// TIA Portal V18 export
FUNCTION_BLOCK "02_Safety_Door"   // FB5, F_LAD
{ S7_Optimized_Access := 'TRUE' }
   VAR_INPUT
      Bypass_For_Commissioning : Bool;
      DIAG : Bool := TRUE;
      CH1 : Bool := TRUE;
      CH2 : Bool := TRUE;
      "Sorter_Running_from MSC" : Bool;
      Sorter_Stop_from_Encoder : Bool;
      Open_Request : Bool;
      Alarm_Filter : Bool;
      Sorter_Door : Bool := TRUE;   // If =1 sorter door management, if =0 management via ESTOP
      ACK_NEC : Bool := TRUE;   // If =1 door need to be reset, if = 0 door will autoreset
      ACK : Bool;
      ON_Lamp : Bool := TRUE;   // If = 1 reset lamp management, if = 0 reset lamp not present
   END_VAR
   VAR_OUTPUT
      Solenoid : Bool;
      EM_Cut : Bool;
      EM_Cut_Delay : Bool;
      Diag_Open : Bool;
      Diag_Alarm : Bool;
      Reset_Lamp : Bool;
   END_VAR
   VAR
      "E-STOP" : ESTOP1;
      TON_Alarm : TON;
      TOF_DoorLamp : TOF;
   END_VAR
   VAR_TEMP
      Alarm_Temp : Bool;
      t_ALARM : Bool;
      t_Lamp : Bool;
   END_VAR
   VAR CONSTANT
      Blink_Cycle_Time : Time := T#1S_260MS;
      ON_Time : Time := T#630MS;
   END_VAR
BEGIN

REGION Network 1: Emergency cut
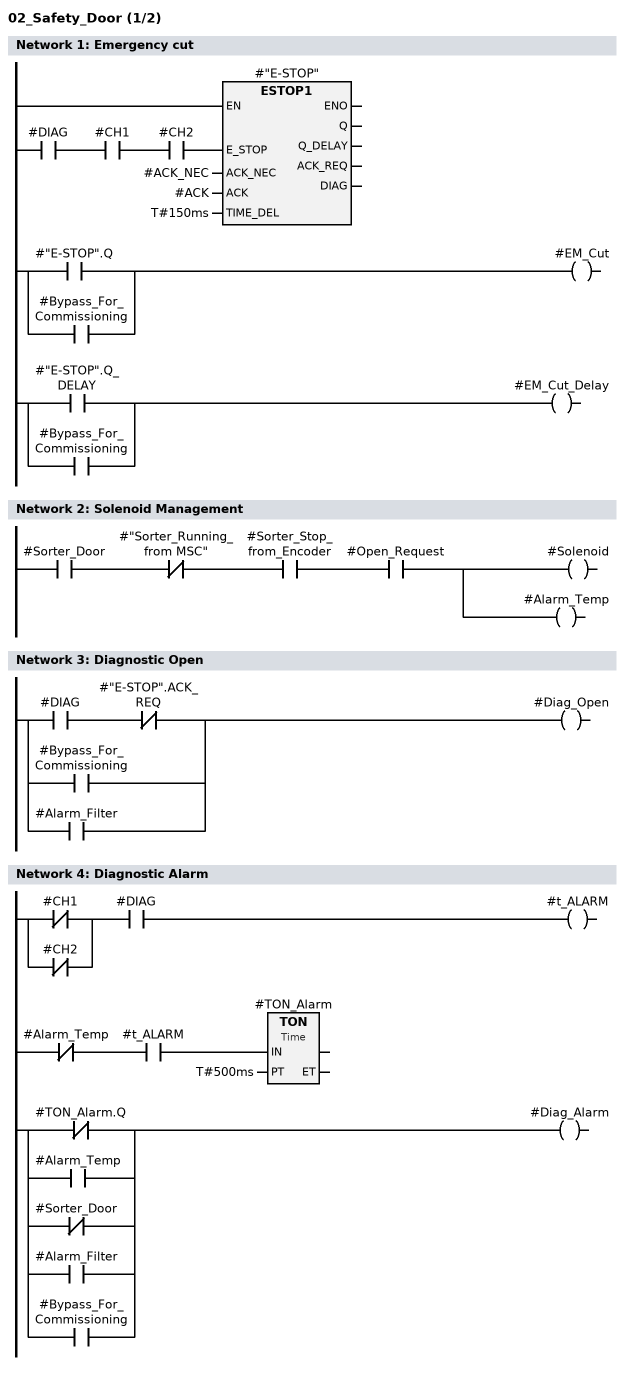
   RUNG wire#powerrail
      #"E-STOP".ESTOP1(E_STOP := wire#w1, ACK_NEC := #ACK_NEC, ACK := #ACK, TIME_DEL := T#150ms, Q =>, Q_DELAY =>, ACK_REQ =>, DIAG =>)
   END_RUNG
   RUNG wire#powerrail
      Contact( #DIAG )
      Contact( #CH1 )
      Contact( #CH2 )
   END_RUNG wire#w1
   RUNG wire#powerrail
      Contact( #"E-STOP".Q )
      wire#w2
      Coil( #EM_Cut )
   END_RUNG
   RUNG wire#powerrail
      Contact( #Bypass_For_Commissioning )
   END_RUNG wire#w2
   RUNG wire#powerrail
      Contact( #"E-STOP".Q_DELAY )
      wire#w3
      Coil( #EM_Cut_Delay )
   END_RUNG
   RUNG wire#powerrail
      Contact( #Bypass_For_Commissioning )
   END_RUNG wire#w3
   // the same network as SCL:
   #"E-STOP"(E_STOP := #DIAG AND #CH1 AND #CH2, ACK_NEC := #ACK_NEC, ACK := #ACK, TIME_DEL := T#150ms);   // ESTOP1
   #EM_Cut := #"E-STOP".Q OR #Bypass_For_Commissioning;
   #EM_Cut_Delay := #"E-STOP".Q_DELAY OR #Bypass_For_Commissioning;
END_REGION

REGION Network 2: Solenoid Management
   RUNG wire#powerrail
      Contact( #Sorter_Door )
      I_Contact( #"Sorter_Running_from MSC" )
      Contact( #Sorter_Stop_from_Encoder )
      Contact( #Open_Request )
      wire#w1
      Coil( #Solenoid )
   END_RUNG
   RUNG wire#w1
      Coil( #Alarm_Temp )
   END_RUNG
   // the same network as SCL:
   #Solenoid := #Sorter_Door AND NOT #"Sorter_Running_from MSC" AND #Sorter_Stop_from_Encoder AND #Open_Request;
   #Alarm_Temp := #Solenoid;
END_REGION

REGION Network 3: Diagnostic Open
   RUNG wire#powerrail
      Contact( #DIAG )
      I_Contact( #"E-STOP".ACK_REQ )
      wire#w1
      Coil( #Diag_Open )
   END_RUNG
   RUNG wire#powerrail
      Contact( #Bypass_For_Commissioning )
   END_RUNG wire#w1
   RUNG wire#powerrail
      Contact( #Alarm_Filter )
   END_RUNG wire#w1
   // the same network as SCL:
   #Diag_Open := (#DIAG AND NOT #"E-STOP".ACK_REQ) OR #Bypass_For_Commissioning OR #Alarm_Filter;
END_REGION

REGION Network 4: Diagnostic Alarm
   RUNG wire#powerrail
      I_Contact( #CH1 )
      wire#w1
      Contact( #DIAG )
      Coil( #t_ALARM )
   END_RUNG
   RUNG wire#powerrail
      I_Contact( #CH2 )
   END_RUNG wire#w1
   RUNG wire#powerrail
      I_Contact( #Alarm_Temp )
      Contact( #t_ALARM )
      { S7_Templates := "[time_type := Time, codedbool_type := DInt]" } #TON_Alarm.TON(pt := T#500ms, et =>)
   END_RUNG
   RUNG wire#powerrail
      I_Contact( #TON_Alarm.Q )
      wire#w2
      Coil( #Diag_Alarm )
   END_RUNG
   RUNG wire#powerrail
      Contact( #Alarm_Temp )
   END_RUNG wire#w2
   RUNG wire#powerrail
      I_Contact( #Sorter_Door )
   END_RUNG wire#w2
   RUNG wire#powerrail
      Contact( #Alarm_Filter )
   END_RUNG wire#w2
   RUNG wire#powerrail
      Contact( #Bypass_For_Commissioning )
   END_RUNG wire#w2
   // the same network as SCL:
   #t_ALARM := (NOT #CH1 OR NOT #CH2) AND #DIAG;
   #TON_Alarm.TON(IN := NOT #Alarm_Temp AND #t_ALARM, PT := T#500ms);
   #Diag_Alarm := NOT #TON_Alarm.Q OR #Alarm_Temp OR NOT #Sorter_Door OR #Alarm_Filter OR #Bypass_For_Commissioning;
END_REGION

REGION Network 5: Rest Lamp
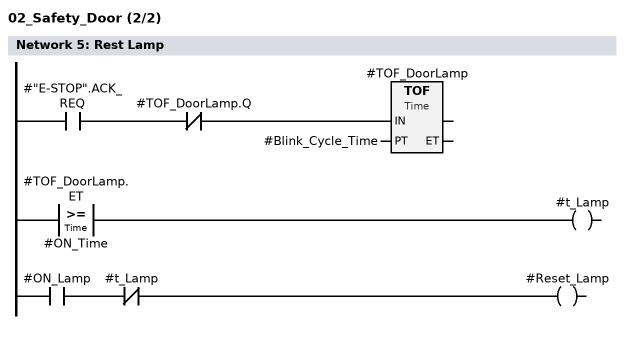
   RUNG wire#powerrail
      Contact( #"E-STOP".ACK_REQ )
      I_Contact( #TOF_DoorLamp.Q )
      { S7_Templates := "[time_type := Time, codedbool_type := DInt]" } #TOF_DoorLamp.TOF(pt := #Blink_Cycle_Time, et =>)
   END_RUNG
   RUNG wire#powerrail
      { S7_Templates := "SrcType := Time" } GE_Contact(in1 := #TOF_DoorLamp.ET, in2 := #ON_Time)
      Coil( #t_Lamp )
   END_RUNG
   RUNG wire#powerrail
      Contact( #ON_Lamp )
      I_Contact( #t_Lamp )
      Coil( #Reset_Lamp )
   END_RUNG
   // the same network as SCL:
   #TOF_DoorLamp.TOF(IN := #"E-STOP".ACK_REQ AND NOT #TOF_DoorLamp.Q, PT := #Blink_Cycle_Time);
   #t_Lamp := #TOF_DoorLamp.ET >= #ON_Time;
   #Reset_Lamp := #ON_Lamp AND NOT #t_Lamp;
END_REGION
END_FUNCTION_BLOCK
